Fanuc KAREL source: IO0035.KL

-- PROVISIONAL review KL for V1013-1; original PC SHA256 6de22c105c02e63815daf236255d5f0687a362baee0cf8f1fdcf881b906d0a04
-- Incomplete behavior may be omitted. Consult companion uncertainty JSON. Do not deploy.
PROGRAM IO0035
%NOLOCKGROUP
-- UNRESOLVED_LOCAL_POOL 5 cells at code offset 13; source declarations unknown
-- DIRECT_LOCAL_WORD_ACCESS alone does not prove INTEGER, REAL, or BOOLEAN
BEGIN
  -- UNRESOLVED_PC offsets 0-18; opcodes 2B,2C,7B
  -- UNRESOLVED_PC offsets 23-30; opcodes 9D,23
  -- UNRESOLVED_PC offsets 35-49; opcodes 2E,22,9D,33,35
  -- UNRESOLVED_PC offsets 54-61; opcodes 9D,23
  -- UNRESOLVED_PC offsets 66-77; opcodes 2E,23
  -- UNRESOLVED_PC offsets 82-99; opcodes 9D,22,21,33,34,1A
  -- UNRESOLVED_PC offsets 104-108; opcodes 7F
  -- UNRESOLVED_PC offsets 113-117; opcodes 27,AA
  -- UNRESOLVED_PC offsets 122-126; opcodes 7F
END IO0035
